FUNCTION_BLOCK AdsSocket
VAR_INPUT
	bEnable : BOOL;
END_VAR
VAR_OUTPUT
	PrgName : STRING; //descriptive string for the name of the running program
	AmsNetId : T_AmsNetId; //this must be assigned even if it is used for local communication - otherwise socket is not considered valid
	AmsPort : T_AmsPort; //for now, use ADS port 851 for communication
END_VAR
VAR_OUTPUT
	receivingData : AdsData;
	sendingData : AdsData;
	
	readBusy : BOOL;
	readError : BOOL;
	readErrorId : UDINT;
	
	writeBusy : BOOL;
	writeError : BOOL;
	writeErrorId : UDINT;
	
	writeReady : BOOL;
	
	timeout : BOOL;
	prevMsgTimestamp : TIMESTRUCT;
END_VAR
VAR	
	targetSocket : STRING := CONCAT('COM.adsMajorNetwork.', localPrgName); //write into the recipient's allocated socket for this system
	adsWriteSymbol : FB_WriteAdsSymByName;
	adsReadSymbol : FB_ReadAdsSymByName;
END_VAR
VAR	
	toggleBit : BOOL; //remote system toggles this bit - use as heartbeat input
	sendingBit : BOOL; //this system toggles this bit - write to remote system's toggleBit
	
	heartbeat : Watchdog;
	writeDelayTimer : TON;
	
	flagWriter : FB_WriteAdsSymByName;
	nameWriter : FB_WriteAdsSymByName;
	netIdWriter : FB_WriteAdsSymByName;
	portWriter : FB_WriteAdsSymByName;
	
	writeSync : BOOL := FALSE;
END_VAR
VAR_STAT
	fbGetLocalAmsNetId : FB_GetLocalAmsNetId;
	
	localPrgName : STRING := TO_STRING(AreaEnum.AREA_2);
	localAmsNetId : T_AmsNetId := '';
	localAmsPort : T_AmsPort := 851;
	
	writeSpacing : TIME := T#200MS;
END_VAR
(*
TCP-style ADS connection that only writes to a buffer in the recipient's AdsTcpUnit module
*)

writeDelayTimer(IN:= NOT writeBusy, PT:= writeSpacing, Q=> writeReady, ET=> );

targetSocket := CONCAT('COM.adsMajorNetwork.', localPrgName);

flagSequence();

IF //do not use this socket if invalid
	NOT bEnable OR
	NOT IsValid
THEN
	RETURN;
END_IF

setup();

(*
if timeout, stop all read/write
if data has no contents, do not send
*)
adsReadSymbol.bRead := NOT timeout AND NOT adsReadSymbol.bRead AND adsReadSymbol.sVarName <> '';
adsWriteSymbol.bWrite := 
	NOT timeout AND
	NOT BufferIsEmpty(sendingData.binaryData) AND 
	NOT adsWriteSymbol.bWrite;

blocks();

(*
IF timeout THEN //stop data read/write attempts
	adsWriteSymbol.bWrite := FALSE;
	adsReadSymbol.bRead := FALSE;
	
ELSE //only writes if data has contents, otherwise remains false
	adsWriteSymbol.bWrite := NOT BufferIsEmpty(sendingData.binaryData) AND NOT adsWriteSymbol.bWrite;
END_IF
*)

METHOD PRIVATE blocks : BOOL
VAR_INPUT
END_VAR
adsReadSymbol(
	bRead:= , 
	sNetId:= AmsNetId, 
	nPort:= AmsPort, 
	sVarName:= , 
	nDestAddr:= , 
	nLen:= , 
	tTimeout:= , 
	eComMode:= , 
	bClearOnError:= , 
	bBusy=> readBusy, 
	bError=> readError, 
	nErrorId=> readErrorId);
	
adsWriteSymbol(
	bWrite:= , 
	sNetId:= AmsNetId, 
	nPort:= AmsPort, 
	sVarName:= CONCAT(targetSocket, '.receivingData'), 
	nSrcAddr:= ADR(sendingData), 
	nLen:= SIZEOF(sendingData), 
	tTimeout:= , 
	eComMode:= eAdsComModeSecureCom, 
	bBusy=> writeBusy, 
	bError=> writeError, 
	nErrorId=> writeErrorId);
	
IF NOT adsWriteSymbol.bBusy THEN
	MEMSET(ADR(sendingData), 0, SIZEOF(sendingData));
END_IF
END_METHOD

METHOD PRIVATE flagSequence : BOOL
VAR_INPUT
END_VAR
heartbeat(
	enable:= TRUE, 
	toggleBit:= toggleBit, 
	timeoutWidth:= DEFAULT_ADS_TIMEOUT, 
	timeout=> timeout);

prevMsgTimestamp := heartbeat.prevMsgTimestamp;

IF NOT flagWriter.bBusy THEN
	sendingBit := NOT sendingBit;
END_IF
END_METHOD

{attribute 'monitoring' := 'call'}
PROPERTY IsValid : BOOL
GET
IsValid := 
	PrgName <> '' AND
	AmsNetId <> '' AND
	AmsPort <> 0;
END_GET
END_PROPERTY

METHOD send : BOOL
VAR_INPUT
	data : REFERENCE TO AdsData;
END_VAR
sendingData := data;
END_METHOD

METHOD PRIVATE setup : BOOL
VAR_INST
	name : STRING;
END_VAR
fbGetLocalAmsNetId(
	bExecute:= (localAmsNetId = '' OR localAmsNetId = '0.0.0.0.0.0') AND NOT fbGetLocalAmsNetId.bExecute, 
	tTimeOut:= , 
	bBusy=> , 
	bError=> , 
	nErrId=> , 
	AddrString=> localAmsNetId, 
	AddrBytes=> );

writeSync := NOT writeSync;

nameWriter(
	bWrite:= writeSync, 
	sNetId:= AmsNetId, 
	nPort:= AmsPort, 
	sVarName:= CONCAT(targetSocket, '.PrgName'), 
	nSrcAddr:= ADR(localPrgName), 
	nLen:= SIZEOF(localPrgName), 
	tTimeout:= , 
	eComMode:= , 
	bBusy=> , 
	bError=> , 
	nErrorId=> );
	
netIdWriter(
	bWrite:= writeSync, 
	sNetId:= AmsNetId, 
	nPort:= AmsPort, 
	sVarName:= CONCAT(targetSocket, '.AmsNetId'), 
	nSrcAddr:= ADR(localAmsNetId), 
	nLen:= SIZEOF(localAmsNetId), 
	tTimeout:= , 
	eComMode:= , 
	bBusy=> , 
	bError=> , 
	nErrorId=> );
	
portWriter(
	bWrite:= writeSync, 
	sNetId:= AmsNetId, 
	nPort:= AmsPort, 
	sVarName:= CONCAT(targetSocket, '.AmsPort'), 
	nSrcAddr:= ADR(localAmsPort), 
	nLen:= SIZEOF(localAmsPort), 
	tTimeout:= , 
	eComMode:= , 
	bBusy=> , 
	bError=> , 
	nErrorId=> );
	
flagWriter(
	bWrite:= writeSync, 
	sNetId:= AmsNetId, 
	nPort:= AmsPort, 
	sVarName:= CONCAT(targetSocket, '.toggleBit'), 
	nSrcAddr:= ADR(sendingBit), 
	nLen:= SIZEOF(sendingBit), 
	tTimeout:= , 
	eComMode:= , 
	bBusy=> , 
	bError=> , 
	nErrorId=> );
END_METHOD

END_FUNCTION_BLOCK

(* stored: Version 1.1.0.1, ProductVersion 3.1.4024.11
   POU AdsSocket: Id {4b08c35a-5e88-4e7b-a45b-894d0e3f10ba}, SpecialFunc None
   Method blocks: Id {aafa1f89-5424-428c-92a9-eff1fd826f0b}
   Method flagSequence: Id {282d8f86-2a36-4b14-910d-5c0d51c4379e}
   Property IsValid: Id {06919978-c9ca-434b-851a-2a74e573c75a}
   Get Get: Id {8efcfd41-9a2b-4700-922a-0a8ec6cada2f}
   Method send: Id {17359b84-8e84-4f55-9ea9-7b9b4062b4aa}
   Method setup: Id {924e3658-3899-4767-999f-eb1a77052422} *)
